// TIA Portal V15.1 export
// export: Created 2020-06-12T07:35:55.8505859Z, ExportSetting None, DisplayName Totally Integrated Automation Portal, DisplayVersion V15.1, DisplayName TIA Portal Openness, DisplayVersion V15.1, DisplayName STEP 7 Professional, DisplayVersion V15.1, DisplayName STEP 7 Safety, DisplayVersion V15.1, DisplayName WinCC Advanced, DisplayVersion V15.1
FUNCTION "SLAG_call" : Void   // FC175, FBD
TITLE = Slag system
{ S7_Optimized_Access := 'TRUE' }
// stored: SetENOAutomatically False
BEGIN

REGION Network 1: Basic control
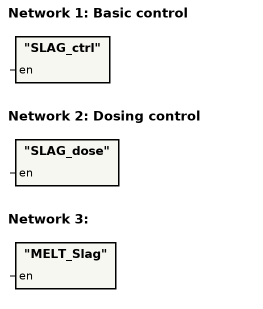
   "SLAG_ctrl"();
END_REGION

REGION Network 2: Dosing control
   "SLAG_dose"();
END_REGION

REGION Network 3
   "MELT_Slag"();
END_REGION
END_FUNCTION
